(* PLC project Tc2_Utilities.HEXSTR_TO_DATA Demo, tc3-libraries-kb TwinCAT 3.1 *)
(* stored: creationDateTime 2026-05-10T19:00:00, modificationDateTime 2026-05-10T19:00:00 *)

PROGRAM P_Demo_HEXSTR_TO_DATA
  VAR
    rResult : UDINT;  (* HEXSTR_TO_DATA 返回值 *)
    bRun : BOOL;  (* 触发一次调用 *)
    sHex : STRING := 'AB CD 01 23';  (* 测试用本地变量 *)
    ar : ARRAY[0..3] OF BYTE;  (* 测试用本地变量 *)
  END_VAR

            // ============================================================
// Tc2_Utilities.HEXSTR_TO_DATA 演示程序（FUNCTION）
// ============================================================
// 验证步骤：
//   1. 引用 Tc2_Utilities
//   2. 编译 + 登录
//   3. 强制 bRun := TRUE 一个周期
//   4. 在线监视 rResult / 各 demo 变量
// ============================================================

IF bRun THEN
    rResult := HEXSTR_TO_DATA(sHex, ADR(ar), SIZEOF(ar));
    bRun := FALSE;
END_IF;

          
END_PROGRAM
